INTERFACE I_Skill_Roboter

METHOD M_Reset : BOOL
VAR_INPUT
END_VAR
END_METHOD

METHOD M_Start : BOOL
VAR_INPUT
END_VAR
END_METHOD

METHOD M_Stop : BOOL
VAR_INPUT
END_VAR
END_METHOD

PROPERTY P_Prozessparameter : sRoboterProzessVariablen
SET
END_SET
END_PROPERTY

PROPERTY P_State : eSkillState
GET
END_GET
END_PROPERTY

END_INTERFACE

(* stored: Version 1.1.0.1
   Itf I_Skill_Roboter: Id {0153326d-f221-4d2a-92c1-c3fc213ce90f}
   Method M_Reset: Id {c4def971-72ce-48b4-a0a4-9fa2acf227ce}
   Method M_Start: Id {8f43df71-bec6-4446-85f5-964246aee3f0}
   Method M_Stop: Id {13b51abf-449f-486d-924e-02b2761140f2}
   Property P_Prozessparameter: Id {ec806130-2d22-478d-b07d-2d2f0af61c71}
   Set Set: Id {40666ce4-1467-48ff-bba6-98ab0bb9df7f}
   Property P_State: Id {c1a99b67-8d9d-4891-b1a2-9533f209fe3d}
   Get Get: Id {f397b8fe-f1e2-4ae9-9c4b-c895c48d8558} *)
